(* CODESYS project Hannover PLC Code.project

Project tree, tasks and I/O mapping:
  Device : CODESYS Control Win V3, 3S - Smart Software Solutions GmbH, order no. 305021, version 3.5.11.30
    application Application
      libraries: Standard, * (System)
      task MainTask (cyclic, interval t#20ms, priority 1) calls PLC_PRG
      program PLC_PRG [ST]
      global variables GVL
      Symbols
      global variables GVL_1
  AC_GENERATOR_DATA
*)

// Device/Application/GVL
{attribute 'qualified_only'}
VAR_GLOBAL


	Mot_Tuer_EGauf: BOOL;
	Mot_Tuer_EGzu: BOOL;
	Tuer_Auf_EG_ES: BOOL;  //Door opened fully
	Tuer_Zu_EG_ES: BOOL;   //Door closed fully
	// Light Baarier Sender
	Li_Tuer_EG: BOOL;
	Tuer_Si_EG: BOOL; // Light Barrier Receiver
	FK_VE_ue_EG: BOOL; // gnd Floor uPPER SWEEP POSITION
	FK_EL_EG: BOOL;  // gnd floor Middle Sweep position 
	FK_VE_un_EG: BOOL; //gnd floor Lowest Sweep position
	Anz_Ruf_EGauf: BOOL;
	In_Anford_EG:BOOL;  //gROUND FLOOR BUTTON
	Anf_EG_FK_Auf: BOOL; //Go uP BUTTON
	Tuer_Auf_EG:BOOL; //Door open ground floor (cONTROL PANEL)
	Tuer_Zu_EG:BOOL;
	Anz_Tuer_EG_Auf:BOOL;
	Anz_Tuer_EG_Zu:BOOL;
	Anz_FK_EG:BOOL;

	Mot_Tuer_1OGauf: BOOL;
	Mot_Tuer_1OGzu: BOOL;
	Tuer_Auf_1OG_ES: BOOL;
	Tuer_Zu_1OG_ES: BOOL;
	// Light Barrier Sender
	Li_Tuer_1OG: BOOL;
	Tuer_Si_1OG: BOOL;  // Light barrier receiver
	FK_VE_ue_1OG: BOOL;   //first Floor uPPER SWEEP POSITION
	FK_EL_1OG: BOOL;       // 1st floor Middle Sweep position 
	FK_VE_un_1OG: BOOL;     //1st floor Lowest Sweep position
	Anz_Ruf_1OGauf: BOOL;
	Anz_Ruf_1OGab: BOOL;
	Anz_1OG_Auf:BOOL;
	Anz_1OG_Ab:BOOL;
	In_Anford_1OG:BOOL;  //fIRST FLOOR BUTTON
	Anf_1OG_FK_Auf: BOOL; //Go uP BUTTON
	Anf_1OG_FK_Ab: BOOL;  //Go down button
	Tuer_Auf_1OG:BOOL;     //dOOr open 1st floor
	Tuer_Zu_1OG:BOOL;       //door closed 1st floor
	Anz_Tuer_1OG_Auf:BOOL;
	Anz_Tuer_1OG_Zu:BOOL;
	Anz_FK_1OG:BOOL;

	Mot_Tuer_2OGauf: BOOL;//
	Mot_Tuer_2OGzu: BOOL;
	Tuer_Auf_2OG_ES: BOOL;
	Tuer_Zu_2OG_ES: BOOL;
	// Light Barrier Sender
	Li_Tuer_2OG: BOOL;
	Tuer_Si_2OG: BOOL; // Light Barrier Receiver
	FK_VE_ue_2OG: BOOL;   //2nd Floor uPPER SWEEP POSITION
	FK_EL_2OG: BOOL;       // 2nd floor Middle Sweep position 
	FK_VE_un_2OG: BOOL;     //2nd floor Lowest Sweep position
	Anz_Ruf_2OGauf: BOOL;
	Anz_Ruf_2OGab: BOOL;
	Anz_2OG_Auf:BOOL;
	Anz_2OG_Ab:BOOL;
	In_Anford_2OG:BOOL;   //2ND FLOOR BUTTON
	Anf_2OG_FK_Auf: BOOL;   //Go uP BUTTON
	Anf_2OG_FK_Ab: BOOL;     //Go down BUTTON
	Tuer_Auf_2OG:BOOL;        //door open 2nd floor
	Tuer_Zu_2OG:BOOL;         //door closed 2nd floor
	Anz_Tuer_2OG_Auf:BOOL;
	Anz_Tuer_2OG_Zu:BOOL;
	Anz_FK_2OG:BOOL;

	Mot_Tuer_3OGauf: BOOL;
	Mot_Tuer_3OGzu: BOOL;
	Mot_Tuer_zu_3OG_man_sim: BOOL;
	Tuer_Auf_3OG_ES: BOOL; //Door opened fully
	Tuer_Zu_3OG_ES: BOOL; //Door closed fully
	// Light Barrier Sender
	Li_Tuer_3OG: BOOL;
	Tuer_Si_3OG: BOOL;  // Light barrier receiver
	FK_VE_ue_3OG: BOOL;   //3rd Floor uPPER SWEEP POSITION
	FK_EL_3OG: BOOL;       // 3rd floor Middle Sweep position
	FK_VE_un_3OG: BOOL;    //3rd floor Lowest Sweep position
	Anz_Ruf_3OGab: BOOL;
	In_Anford_3OG:BOOL;   //3RD FLOOR BUTTON
	Anf_3OG_FK_Ab: BOOL;  //Go uP down
	Tuer_Auf_3OG:BOOL;    //door open 3rd floor
	Tuer_Zu_3OG:BOOL;      //door closed 3rd floor    
	Anz_Tuer_3OG_Auf:BOOL;
	Anz_Tuer_3OG_Zu:BOOL;
	Anz_FK_3OG:BOOL;


	Mot_FK_Auf: BOOL;
	Mot_FK_Ab: BOOL;
	Fahrk_Auf:BOOL; //Car Open
	Fahrk_Ab:BOOL;  //CAR CLOSE
	Ue_Last:BOOL;  //Car Overload
	Anz_FK_Auf:BOOL;
	Anz_FK_Ab:BOOL;
	Anz_FK_zuhoch:BOOL;
	Anz_FK_zutief:BOOL;

	Tuer_Auf:BOOL; //Open the door
	NOTRUF: BOOL; //Emergency Csll
	IN_Steu_Ein: BOOL;  //Interior Controls
	Not_Aus:BOOL:=TRUE; //Emergency Stop Switch
	Betr_Art_Prog:BOOL;
	Anz_Prog:BOOL;
	Anz_Insp:BOOL;
	Anz_InnenST:BOOL;
	Anz_NOT_AUS_BP:BOOL;
	Anz_NOT_AUS_FK:BOOL;
	Lamp_Test:BOOL;
	Anf_Rel: BOOL;



	//INT_Bewegung_Stockwerke: INTEGRAL;
	Bewegung_Stockwerke_Visu: REAL;
	Bewegung_Stockwerke_inv:REAL;

	PROG:BOOL;
	Betriebsart:BOOL:=TRUE;  // program operation /Start
	PROG_Visu:BOOL;

	Hindernis_EG_sim: BOOL; //obstacle at gnd floor
	Hindernis_1OG_sim: BOOL; //obstacle at first floot
	Hindernis_2OG_sim: BOOL; //obstacle at 2nd floor
	Hindernis_3OG_sim: BOOL;  //obstacle at 3rd floor
END_VAR

// Device/Application/GVL_1
{attribute 'qualified_only'}
VAR_GLOBAL
	MOTOR1: BOOL := FALSE;
	BUTTON1: BOOL := FALSE;
END_VAR

// Device/Application/PLC_PRG
PROGRAM PLC_PRG
VAR
END_VAR

IF GVL_1.BUTTON1 THEN
	GVL_1.MOTOR1 := TRUE;
END_IF

END_PROGRAM
